PROGRAM PRG_PAOL_02_LightboxScanersCtrl
VAR

	tonEnableCameraSystem				: TON;
	bEnablePackAggregationCameraSystem	: BOOL;
	bEnablePackTriggeringAfterDelayON		: BOOL;

	tofPackAggregationCameraOFFDelay 		: TOF;
	bEnablePackTriggeringAfterDelayOFF		: BOOL;

	fbLightboxLensAirPuls				: FB_Puls;
	tonLightboxLensAirNextBlow		: TON;
	rtrigLightboxLensAirBlowing		: R_TRIG;
	tonLightboxLensAirBlowing		: TOF;
	bPackAggregCameraTrig4Enable			: BOOL;

	fbCameraBoxRead					: FB_3CAM_CameraBoxRead;


	bCameraTriggersArmed			: BOOL;
	bCameraTrigger1Conditioned		: BOOL;
	bCameraTrigger2Conditioned		: BOOL;
	bCameraTrigger3Conditioned		: BOOL;
	bCameraTrigger4Conditioned		: BOOL;

	rtrigCameraTrigger					: ARRAY[0..4] OF R_TRIG;
	aCameraTrigger					: ARRAY[0..4] OF BOOL;
	fbCameraSequenceNo				: FB_3CAM_CameraSequenceNo;

	fbPackScanners_2x5Packs			: FB_3CAM_PackScanners2x5Packs;
	fbPackScanners_3x4Packs			: FB_3CAM_PackScanners3x4Packs;
	fbPackScanners_4x3Packs			: FB_3CAM_PackScanners4x3Packs;
	fbSelectCameraMap				: FB_3CAM_SelectCameraMap;


	fbOUTER_AddNewTriggerID		: FB_PAOL_AddNewTriggerID;
	fbMoveOuterStatusArray			: FB_PACK_MoveOuterStatusArray;	(*Actually is moving OCVPackStatusArray*)

	aPackScanner						: ARRAY[1..3] OF ST_SCANNER_CameraMap;
	fbScannerCtrl						: ARRAY[1..3] OF FB_SCANNER_CameraSelect;
	fbPackCameraEvaluation			: ARRAY[1..3] OF FB_SCANNER_Evaluation;

	fbAddPackCodes					: ARRAY[1..3] OF FB_3CAM_AddPackCodes;

	fbInfeedCamerasSync 				: ARRAY[1..3] OF FB_PAOL_InfeedCamerasSync;

	tonDelayStopOuter					: TON;
	bCameraBufferHighTest 			: BOOL;

	bPackCodeDataInvalid				: BOOL;
	ctuConsecutiveDataInvalid		: CTU;
END_VAR
VAR // added by the converter: edge detectors and wires of the graphical bodies
    _w1, _w3 : BOOL;
    _w2 : UDINT;
END_VAR

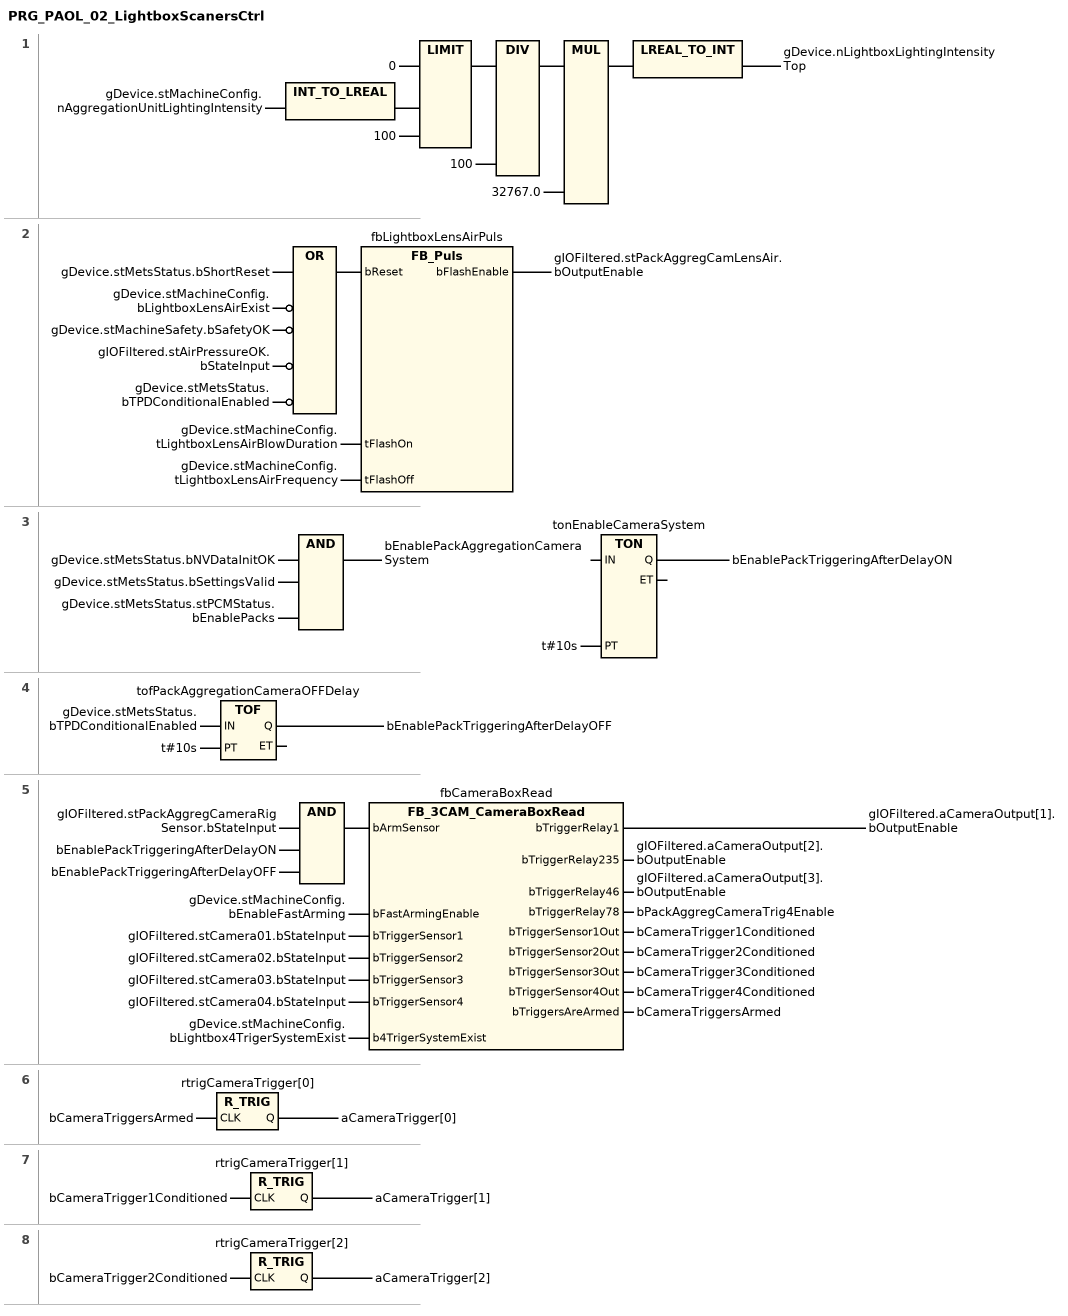
// NETWORK 1
gDevice.nLightboxLightingIntensityTop := LREAL_TO_INT((LIMIT(0, INT_TO_LREAL(gDevice.stMachineConfig.nAggregationUnitLightingIntensity), 100) / 100) * 32767.0);

// NETWORK 2
fbLightboxLensAirPuls(
    bReset := gDevice.stMetsStatus.bShortReset OR NOT gDevice.stMachineConfig.bLightboxLensAirExist OR NOT gDevice.stMachineSafety.bSafetyOK OR NOT gIOFiltered.stAirPressureOK.bStateInput OR NOT gDevice.stMetsStatus.bTPDConditionalEnabled,
    tFlashOn := gDevice.stMachineConfig.tLightboxLensAirBlowDuration,
    tFlashOff := gDevice.stMachineConfig.tLightboxLensAirFrequency); // FB_Puls
gIOFiltered.stPackAggregCamLensAir.bOutputEnable := fbLightboxLensAirPuls.bFlashEnable;

// NETWORK 3
_w1 := gDevice.stMetsStatus.bNVDataInitOK AND gDevice.stMetsStatus.bSettingsValid AND gDevice.stMetsStatus.stPCMStatus.bEnablePacks;
bEnablePackAggregationCameraSystem := _w1;
tonEnableCameraSystem(IN := _w1, PT := t#10s); // TON
bEnablePackTriggeringAfterDelayON := tonEnableCameraSystem.Q;

// NETWORK 4
tofPackAggregationCameraOFFDelay(IN := gDevice.stMetsStatus.bTPDConditionalEnabled, PT := t#10s); // TOF
bEnablePackTriggeringAfterDelayOFF := tofPackAggregationCameraOFFDelay.Q;

// NETWORK 5
fbCameraBoxRead(
    bArmSensor := gIOFiltered.stPackAggregCameraRigSensor.bStateInput AND bEnablePackTriggeringAfterDelayON AND bEnablePackTriggeringAfterDelayOFF,
    bFastArmingEnable := gDevice.stMachineConfig.bEnableFastArming,
    bTriggerSensor1 := gIOFiltered.stCamera01.bStateInput,
    bTriggerSensor2 := gIOFiltered.stCamera02.bStateInput,
    bTriggerSensor3 := gIOFiltered.stCamera03.bStateInput,
    bTriggerSensor4 := gIOFiltered.stCamera04.bStateInput,
    b4TrigerSystemExist := gDevice.stMachineConfig.bLightbox4TrigerSystemExist,
    bTriggerRelay235 => gIOFiltered.aCameraOutput[2].bOutputEnable,
    bTriggerRelay46 => gIOFiltered.aCameraOutput[3].bOutputEnable,
    bTriggerRelay78 => bPackAggregCameraTrig4Enable,
    bTriggerSensor1Out => bCameraTrigger1Conditioned,
    bTriggerSensor2Out => bCameraTrigger2Conditioned,
    bTriggerSensor3Out => bCameraTrigger3Conditioned,
    bTriggerSensor4Out => bCameraTrigger4Conditioned,
    bTriggersAreArmed => bCameraTriggersArmed); // FB_3CAM_CameraBoxRead
gIOFiltered.aCameraOutput[1].bOutputEnable := fbCameraBoxRead.bTriggerRelay1;

// NETWORK 6
rtrigCameraTrigger[0](CLK := bCameraTriggersArmed); // R_TRIG
aCameraTrigger[0] := rtrigCameraTrigger[0].Q;

// NETWORK 7
rtrigCameraTrigger[1](CLK := bCameraTrigger1Conditioned); // R_TRIG
aCameraTrigger[1] := rtrigCameraTrigger[1].Q;

// NETWORK 8
rtrigCameraTrigger[2](CLK := bCameraTrigger2Conditioned); // R_TRIG
aCameraTrigger[2] := rtrigCameraTrigger[2].Q;

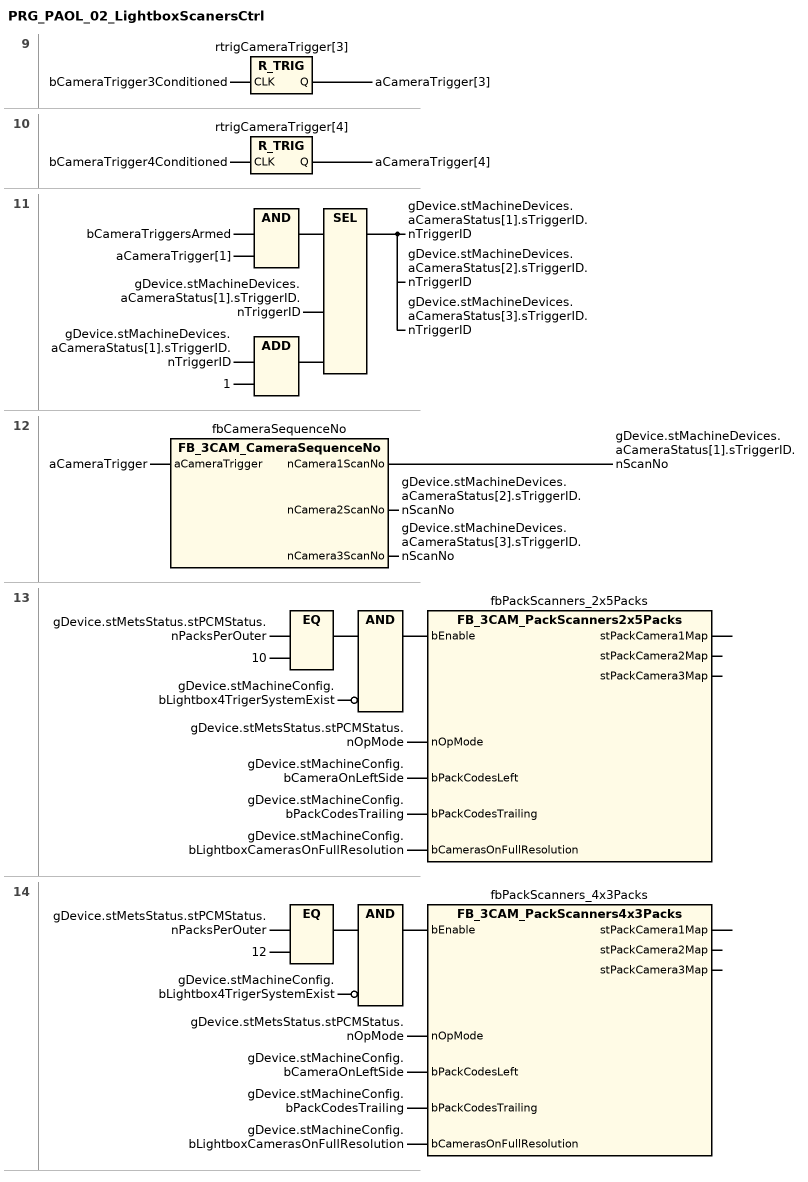
// NETWORK 9
rtrigCameraTrigger[3](CLK := bCameraTrigger3Conditioned); // R_TRIG
aCameraTrigger[3] := rtrigCameraTrigger[3].Q;

// NETWORK 10
rtrigCameraTrigger[4](CLK := bCameraTrigger4Conditioned); // R_TRIG
aCameraTrigger[4] := rtrigCameraTrigger[4].Q;

// NETWORK 11
_w2 := SEL(bCameraTriggersArmed AND aCameraTrigger[1], gDevice.stMachineDevices.aCameraStatus[1].sTriggerID.nTriggerID, gDevice.stMachineDevices.aCameraStatus[1].sTriggerID.nTriggerID + 1);
gDevice.stMachineDevices.aCameraStatus[1].sTriggerID.nTriggerID := _w2;
gDevice.stMachineDevices.aCameraStatus[2].sTriggerID.nTriggerID := _w2;
gDevice.stMachineDevices.aCameraStatus[3].sTriggerID.nTriggerID := _w2;

// NETWORK 12
fbCameraSequenceNo(
    aCameraTrigger := aCameraTrigger,
    nCamera2ScanNo => gDevice.stMachineDevices.aCameraStatus[2].sTriggerID.nScanNo,
    nCamera3ScanNo => gDevice.stMachineDevices.aCameraStatus[3].sTriggerID.nScanNo); // FB_3CAM_CameraSequenceNo
gDevice.stMachineDevices.aCameraStatus[1].sTriggerID.nScanNo := fbCameraSequenceNo.nCamera1ScanNo;

// NETWORK 13
fbPackScanners_2x5Packs(
    bEnable := gDevice.stMetsStatus.stPCMStatus.nPacksPerOuter = 10 AND NOT gDevice.stMachineConfig.bLightbox4TrigerSystemExist,
    nOpMode := gDevice.stMetsStatus.stPCMStatus.nOpMode,
    bPackCodesLeft := gDevice.stMachineConfig.bCameraOnLeftSide,
    bPackCodesTrailing := gDevice.stMachineConfig.bPackCodesTrailing,
    bCamerasOnFullResolution := gDevice.stMachineConfig.bLightboxCamerasOnFullResolution); // FB_3CAM_PackScanners2x5Packs

// NETWORK 14
fbPackScanners_4x3Packs(
    bEnable := gDevice.stMetsStatus.stPCMStatus.nPacksPerOuter = 12 AND NOT gDevice.stMachineConfig.bLightbox4TrigerSystemExist,
    nOpMode := gDevice.stMetsStatus.stPCMStatus.nOpMode,
    bPackCodesLeft := gDevice.stMachineConfig.bCameraOnLeftSide,
    bPackCodesTrailing := gDevice.stMachineConfig.bPackCodesTrailing,
    bCamerasOnFullResolution := gDevice.stMachineConfig.bLightboxCamerasOnFullResolution); // FB_3CAM_PackScanners4x3Packs

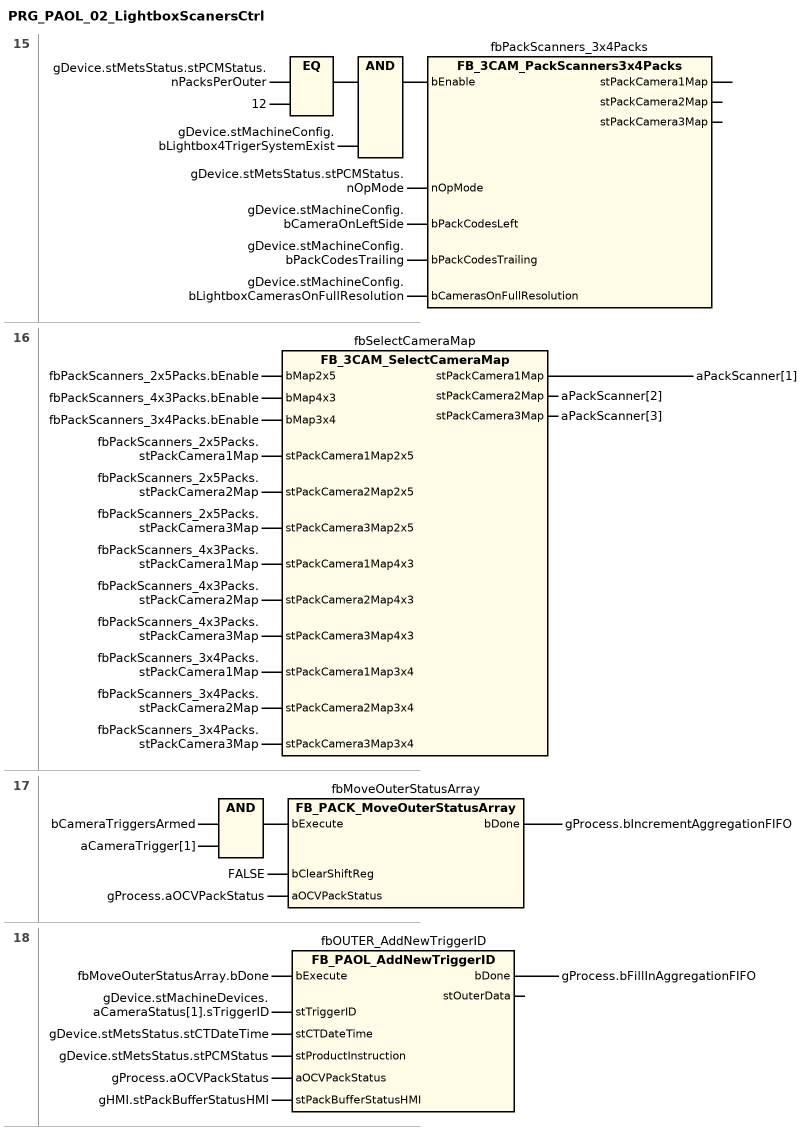
// NETWORK 15
fbPackScanners_3x4Packs(
    bEnable := gDevice.stMetsStatus.stPCMStatus.nPacksPerOuter = 12 AND gDevice.stMachineConfig.bLightbox4TrigerSystemExist,
    nOpMode := gDevice.stMetsStatus.stPCMStatus.nOpMode,
    bPackCodesLeft := gDevice.stMachineConfig.bCameraOnLeftSide,
    bPackCodesTrailing := gDevice.stMachineConfig.bPackCodesTrailing,
    bCamerasOnFullResolution := gDevice.stMachineConfig.bLightboxCamerasOnFullResolution); // FB_3CAM_PackScanners3x4Packs

// NETWORK 16
fbSelectCameraMap(
    bMap2x5 := fbPackScanners_2x5Packs.bEnable,
    bMap4x3 := fbPackScanners_4x3Packs.bEnable,
    bMap3x4 := fbPackScanners_3x4Packs.bEnable,
    stPackCamera1Map2x5 := fbPackScanners_2x5Packs.stPackCamera1Map,
    stPackCamera2Map2x5 := fbPackScanners_2x5Packs.stPackCamera2Map,
    stPackCamera3Map2x5 := fbPackScanners_2x5Packs.stPackCamera3Map,
    stPackCamera1Map4x3 := fbPackScanners_4x3Packs.stPackCamera1Map,
    stPackCamera2Map4x3 := fbPackScanners_4x3Packs.stPackCamera2Map,
    stPackCamera3Map4x3 := fbPackScanners_4x3Packs.stPackCamera3Map,
    stPackCamera1Map3x4 := fbPackScanners_3x4Packs.stPackCamera1Map,
    stPackCamera2Map3x4 := fbPackScanners_3x4Packs.stPackCamera2Map,
    stPackCamera3Map3x4 := fbPackScanners_3x4Packs.stPackCamera3Map,
    stPackCamera2Map => aPackScanner[2],
    stPackCamera3Map => aPackScanner[3]); // FB_3CAM_SelectCameraMap
aPackScanner[1] := fbSelectCameraMap.stPackCamera1Map;

// NETWORK 17
fbMoveOuterStatusArray(
    bExecute := bCameraTriggersArmed AND aCameraTrigger[1],
    bClearShiftReg := FALSE,
    aOCVPackStatus := gProcess.aOCVPackStatus); // FB_PACK_MoveOuterStatusArray
gProcess.bIncrementAggregationFIFO := fbMoveOuterStatusArray.bDone;

// NETWORK 18
fbOUTER_AddNewTriggerID(
    bExecute := fbMoveOuterStatusArray.bDone,
    stTriggerID := gDevice.stMachineDevices.aCameraStatus[1].sTriggerID,
    stCTDateTime := gDevice.stMetsStatus.stCTDateTime,
    stProductInstruction := gDevice.stMetsStatus.stPCMStatus,
    aOCVPackStatus := gProcess.aOCVPackStatus,
    stPackBufferStatusHMI := gHMI.stPackBufferStatusHMI); // FB_PAOL_AddNewTriggerID
gProcess.bFillInAggregationFIFO := fbOUTER_AddNewTriggerID.bDone;

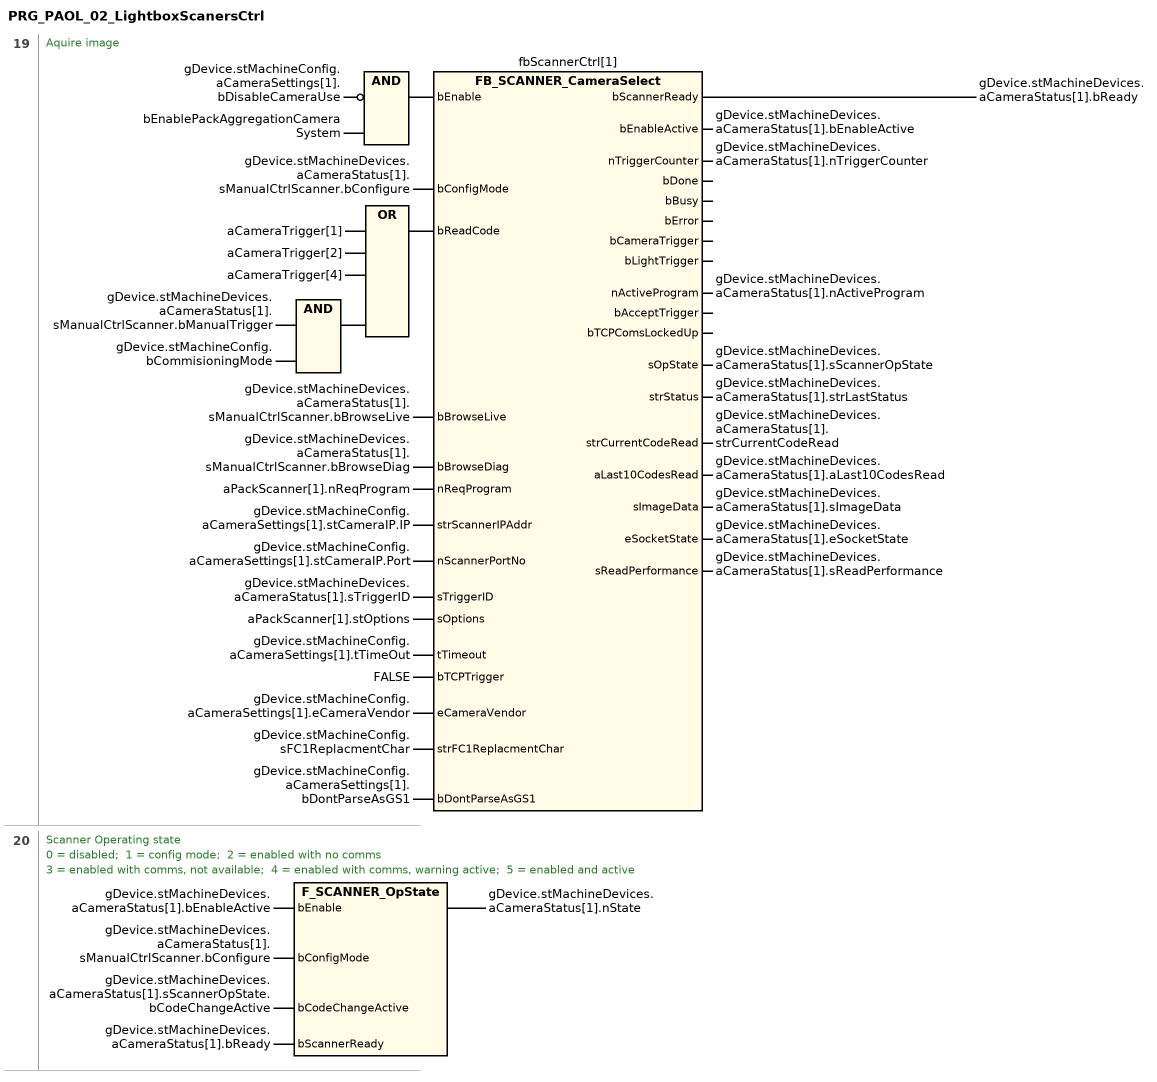
// NETWORK 19
// Aquire image
fbScannerCtrl[1](
    bEnable := NOT gDevice.stMachineConfig.aCameraSettings[1].bDisableCameraUse AND bEnablePackAggregationCameraSystem,
    bConfigMode := gDevice.stMachineDevices.aCameraStatus[1].sManualCtrlScanner.bConfigure,
    bReadCode := aCameraTrigger[1] OR aCameraTrigger[2] OR aCameraTrigger[4] OR gDevice.stMachineDevices.aCameraStatus[1].sManualCtrlScanner.bManualTrigger AND gDevice.stMachineConfig.bCommisioningMode,
    bBrowseLive := gDevice.stMachineDevices.aCameraStatus[1].sManualCtrlScanner.bBrowseLive,
    bBrowseDiag := gDevice.stMachineDevices.aCameraStatus[1].sManualCtrlScanner.bBrowseDiag,
    nReqProgram := aPackScanner[1].nReqProgram,
    strScannerIPAddr := gDevice.stMachineConfig.aCameraSettings[1].stCameraIP.IP,
    nScannerPortNo := gDevice.stMachineConfig.aCameraSettings[1].stCameraIP.Port,
    sTriggerID := gDevice.stMachineDevices.aCameraStatus[1].sTriggerID,
    sOptions := aPackScanner[1].stOptions,
    tTimeout := gDevice.stMachineConfig.aCameraSettings[1].tTimeOut,
    bTCPTrigger := FALSE,
    eCameraVendor := gDevice.stMachineConfig.aCameraSettings[1].eCameraVendor,
    strFC1ReplacmentChar := gDevice.stMachineConfig.sFC1ReplacmentChar,
    bDontParseAsGS1 := gDevice.stMachineConfig.aCameraSettings[1].bDontParseAsGS1,
    bEnableActive => gDevice.stMachineDevices.aCameraStatus[1].bEnableActive,
    nTriggerCounter => gDevice.stMachineDevices.aCameraStatus[1].nTriggerCounter,
    nActiveProgram => gDevice.stMachineDevices.aCameraStatus[1].nActiveProgram,
    sOpState => gDevice.stMachineDevices.aCameraStatus[1].sScannerOpState,
    strStatus => gDevice.stMachineDevices.aCameraStatus[1].strLastStatus,
    strCurrentCodeRead => gDevice.stMachineDevices.aCameraStatus[1].strCurrentCodeRead,
    aLast10CodesRead => gDevice.stMachineDevices.aCameraStatus[1].aLast10CodesRead,
    sImageData => gDevice.stMachineDevices.aCameraStatus[1].sImageData,
    eSocketState => gDevice.stMachineDevices.aCameraStatus[1].eSocketState,
    sReadPerformance => gDevice.stMachineDevices.aCameraStatus[1].sReadPerformance); // FB_SCANNER_CameraSelect
gDevice.stMachineDevices.aCameraStatus[1].bReady := fbScannerCtrl[1].bScannerReady;

// NETWORK 20
// 					Scanner Operating state
// 0 = disabled;  1 = config mode;  2 = enabled with no comms
// 3 = enabled with comms, not available;  4 = enabled with comms, warning active;  5 = enabled and active
//
gDevice.stMachineDevices.aCameraStatus[1].nState := F_SCANNER_OpState(bEnable := gDevice.stMachineDevices.aCameraStatus[1].bEnableActive, bConfigMode := gDevice.stMachineDevices.aCameraStatus[1].sManualCtrlScanner.bConfigure, bCodeChangeActive := gDevice.stMachineDevices.aCameraStatus[1].sScannerOpState.bCodeChangeActive, bScannerReady := gDevice.stMachineDevices.aCameraStatus[1].bReady);

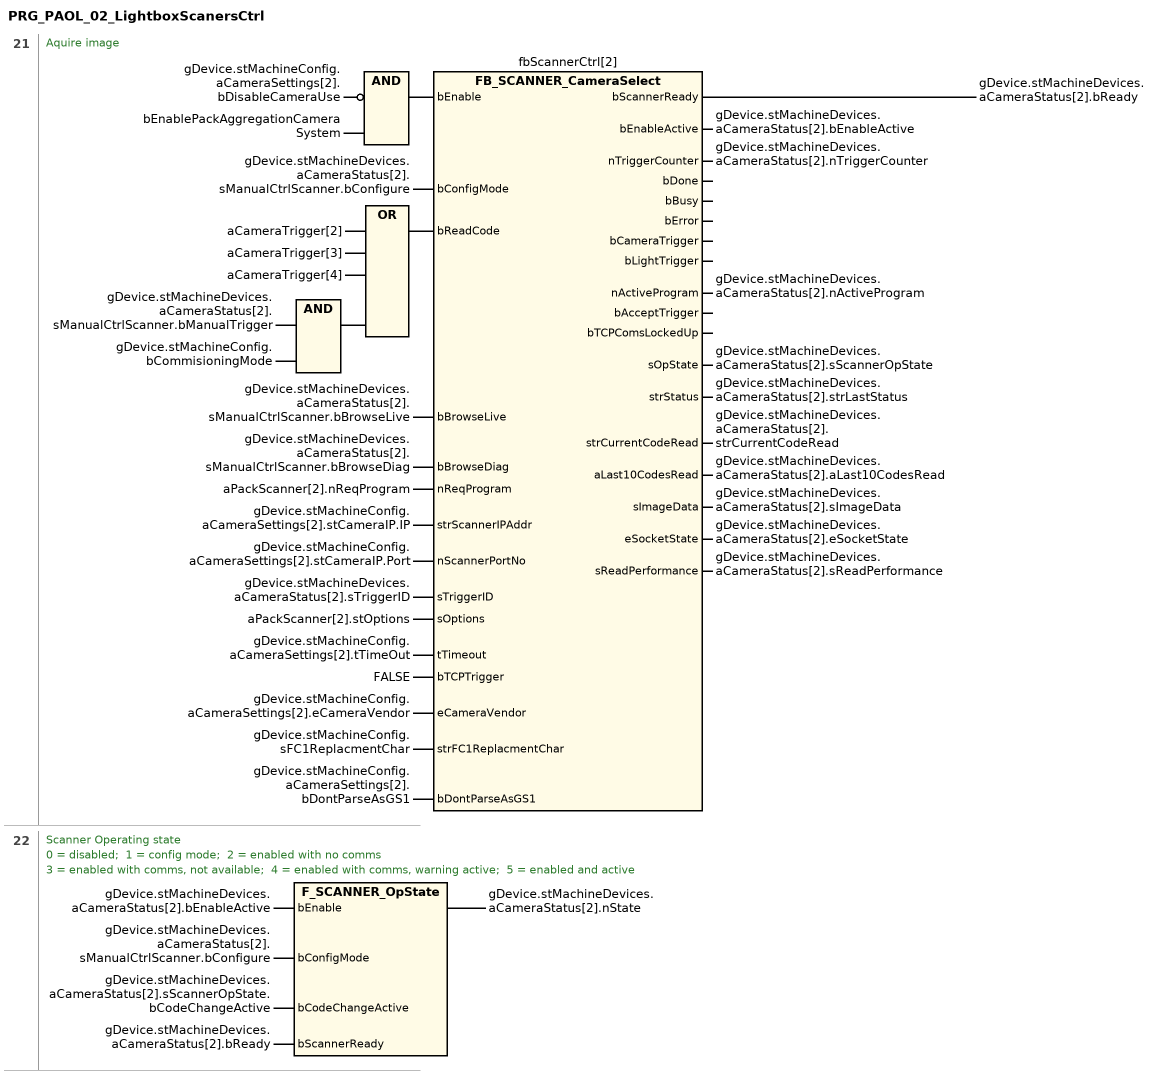
// NETWORK 21
// Aquire image
fbScannerCtrl[2](
    bEnable := NOT gDevice.stMachineConfig.aCameraSettings[2].bDisableCameraUse AND bEnablePackAggregationCameraSystem,
    bConfigMode := gDevice.stMachineDevices.aCameraStatus[2].sManualCtrlScanner.bConfigure,
    bReadCode := aCameraTrigger[2] OR aCameraTrigger[3] OR aCameraTrigger[4] OR gDevice.stMachineDevices.aCameraStatus[2].sManualCtrlScanner.bManualTrigger AND gDevice.stMachineConfig.bCommisioningMode,
    bBrowseLive := gDevice.stMachineDevices.aCameraStatus[2].sManualCtrlScanner.bBrowseLive,
    bBrowseDiag := gDevice.stMachineDevices.aCameraStatus[2].sManualCtrlScanner.bBrowseDiag,
    nReqProgram := aPackScanner[2].nReqProgram,
    strScannerIPAddr := gDevice.stMachineConfig.aCameraSettings[2].stCameraIP.IP,
    nScannerPortNo := gDevice.stMachineConfig.aCameraSettings[2].stCameraIP.Port,
    sTriggerID := gDevice.stMachineDevices.aCameraStatus[2].sTriggerID,
    sOptions := aPackScanner[2].stOptions,
    tTimeout := gDevice.stMachineConfig.aCameraSettings[2].tTimeOut,
    bTCPTrigger := FALSE,
    eCameraVendor := gDevice.stMachineConfig.aCameraSettings[2].eCameraVendor,
    strFC1ReplacmentChar := gDevice.stMachineConfig.sFC1ReplacmentChar,
    bDontParseAsGS1 := gDevice.stMachineConfig.aCameraSettings[2].bDontParseAsGS1,
    bEnableActive => gDevice.stMachineDevices.aCameraStatus[2].bEnableActive,
    nTriggerCounter => gDevice.stMachineDevices.aCameraStatus[2].nTriggerCounter,
    nActiveProgram => gDevice.stMachineDevices.aCameraStatus[2].nActiveProgram,
    sOpState => gDevice.stMachineDevices.aCameraStatus[2].sScannerOpState,
    strStatus => gDevice.stMachineDevices.aCameraStatus[2].strLastStatus,
    strCurrentCodeRead => gDevice.stMachineDevices.aCameraStatus[2].strCurrentCodeRead,
    aLast10CodesRead => gDevice.stMachineDevices.aCameraStatus[2].aLast10CodesRead,
    sImageData => gDevice.stMachineDevices.aCameraStatus[2].sImageData,
    eSocketState => gDevice.stMachineDevices.aCameraStatus[2].eSocketState,
    sReadPerformance => gDevice.stMachineDevices.aCameraStatus[2].sReadPerformance); // FB_SCANNER_CameraSelect
gDevice.stMachineDevices.aCameraStatus[2].bReady := fbScannerCtrl[2].bScannerReady;

// NETWORK 22
// 					Scanner Operating state
// 0 = disabled;  1 = config mode;  2 = enabled with no comms
// 3 = enabled with comms, not available;  4 = enabled with comms, warning active;  5 = enabled and active
//
gDevice.stMachineDevices.aCameraStatus[2].nState := F_SCANNER_OpState(bEnable := gDevice.stMachineDevices.aCameraStatus[2].bEnableActive, bConfigMode := gDevice.stMachineDevices.aCameraStatus[2].sManualCtrlScanner.bConfigure, bCodeChangeActive := gDevice.stMachineDevices.aCameraStatus[2].sScannerOpState.bCodeChangeActive, bScannerReady := gDevice.stMachineDevices.aCameraStatus[2].bReady);

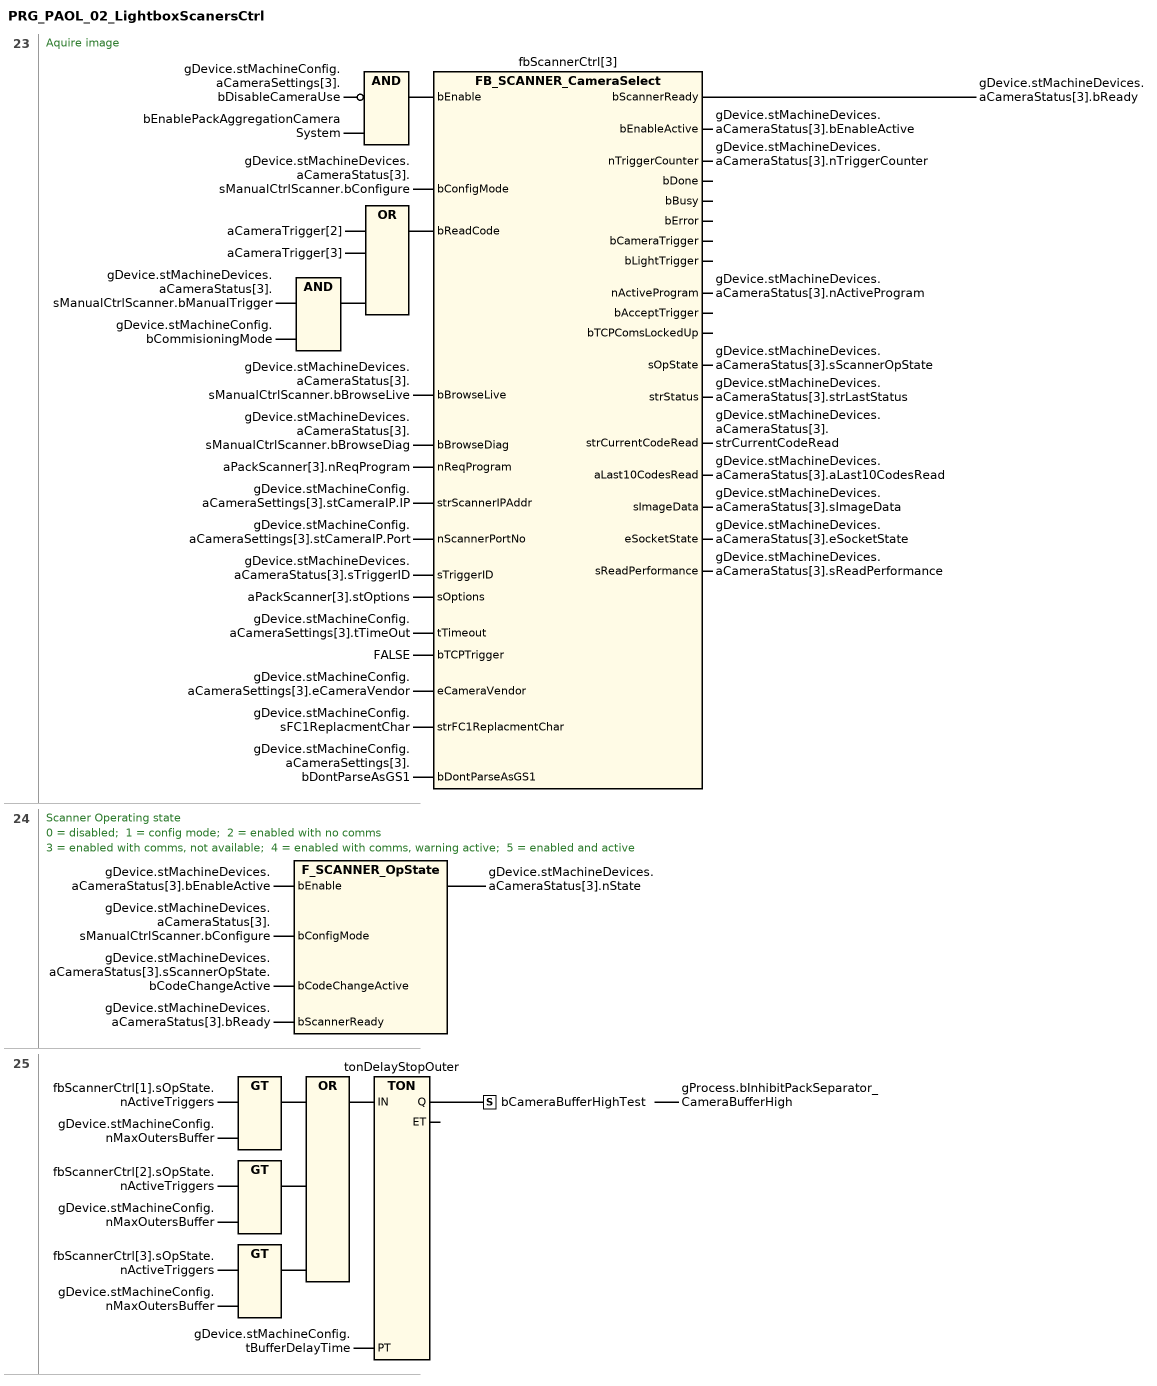
// NETWORK 23
// Aquire image
fbScannerCtrl[3](
    bEnable := NOT gDevice.stMachineConfig.aCameraSettings[3].bDisableCameraUse AND bEnablePackAggregationCameraSystem,
    bConfigMode := gDevice.stMachineDevices.aCameraStatus[3].sManualCtrlScanner.bConfigure,
    bReadCode := aCameraTrigger[2] OR aCameraTrigger[3] OR gDevice.stMachineDevices.aCameraStatus[3].sManualCtrlScanner.bManualTrigger AND gDevice.stMachineConfig.bCommisioningMode,
    bBrowseLive := gDevice.stMachineDevices.aCameraStatus[3].sManualCtrlScanner.bBrowseLive,
    bBrowseDiag := gDevice.stMachineDevices.aCameraStatus[3].sManualCtrlScanner.bBrowseDiag,
    nReqProgram := aPackScanner[3].nReqProgram,
    strScannerIPAddr := gDevice.stMachineConfig.aCameraSettings[3].stCameraIP.IP,
    nScannerPortNo := gDevice.stMachineConfig.aCameraSettings[3].stCameraIP.Port,
    sTriggerID := gDevice.stMachineDevices.aCameraStatus[3].sTriggerID,
    sOptions := aPackScanner[3].stOptions,
    tTimeout := gDevice.stMachineConfig.aCameraSettings[3].tTimeOut,
    bTCPTrigger := FALSE,
    eCameraVendor := gDevice.stMachineConfig.aCameraSettings[3].eCameraVendor,
    strFC1ReplacmentChar := gDevice.stMachineConfig.sFC1ReplacmentChar,
    bDontParseAsGS1 := gDevice.stMachineConfig.aCameraSettings[3].bDontParseAsGS1,
    bEnableActive => gDevice.stMachineDevices.aCameraStatus[3].bEnableActive,
    nTriggerCounter => gDevice.stMachineDevices.aCameraStatus[3].nTriggerCounter,
    nActiveProgram => gDevice.stMachineDevices.aCameraStatus[3].nActiveProgram,
    sOpState => gDevice.stMachineDevices.aCameraStatus[3].sScannerOpState,
    strStatus => gDevice.stMachineDevices.aCameraStatus[3].strLastStatus,
    strCurrentCodeRead => gDevice.stMachineDevices.aCameraStatus[3].strCurrentCodeRead,
    aLast10CodesRead => gDevice.stMachineDevices.aCameraStatus[3].aLast10CodesRead,
    sImageData => gDevice.stMachineDevices.aCameraStatus[3].sImageData,
    eSocketState => gDevice.stMachineDevices.aCameraStatus[3].eSocketState,
    sReadPerformance => gDevice.stMachineDevices.aCameraStatus[3].sReadPerformance); // FB_SCANNER_CameraSelect
gDevice.stMachineDevices.aCameraStatus[3].bReady := fbScannerCtrl[3].bScannerReady;

// NETWORK 24
// 					Scanner Operating state
// 0 = disabled;  1 = config mode;  2 = enabled with no comms
// 3 = enabled with comms, not available;  4 = enabled with comms, warning active;  5 = enabled and active
//
gDevice.stMachineDevices.aCameraStatus[3].nState := F_SCANNER_OpState(bEnable := gDevice.stMachineDevices.aCameraStatus[3].bEnableActive, bConfigMode := gDevice.stMachineDevices.aCameraStatus[3].sManualCtrlScanner.bConfigure, bCodeChangeActive := gDevice.stMachineDevices.aCameraStatus[3].sScannerOpState.bCodeChangeActive, bScannerReady := gDevice.stMachineDevices.aCameraStatus[3].bReady);

// NETWORK 25
tonDelayStopOuter(IN := fbScannerCtrl[1].sOpState.nActiveTriggers > gDevice.stMachineConfig.nMaxOutersBuffer OR fbScannerCtrl[2].sOpState.nActiveTriggers > gDevice.stMachineConfig.nMaxOutersBuffer OR fbScannerCtrl[3].sOpState.nActiveTriggers > gDevice.stMachineConfig.nMaxOutersBuffer, PT := gDevice.stMachineConfig.tBufferDelayTime); // TON
bCameraBufferHighTest S= tonDelayStopOuter.Q;
gProcess.bInhibitPackSeparator_CameraBufferHigh := tonDelayStopOuter.Q;

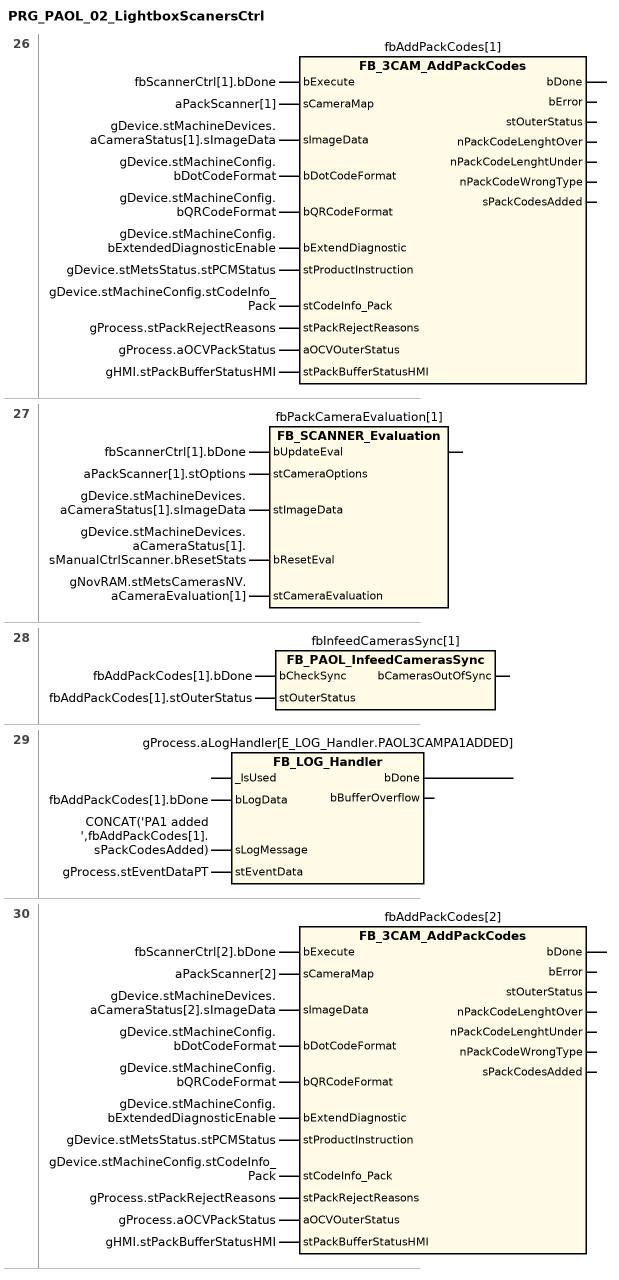
// NETWORK 26
fbAddPackCodes[1](
    bExecute := fbScannerCtrl[1].bDone,
    sCameraMap := aPackScanner[1],
    sImageData := gDevice.stMachineDevices.aCameraStatus[1].sImageData,
    bDotCodeFormat := gDevice.stMachineConfig.bDotCodeFormat,
    bQRCodeFormat := gDevice.stMachineConfig.bQRCodeFormat,
    bExtendDiagnostic := gDevice.stMachineConfig.bExtendedDiagnosticEnable,
    stProductInstruction := gDevice.stMetsStatus.stPCMStatus,
    stCodeInfo_Pack := gDevice.stMachineConfig.stCodeInfo_Pack,
    stPackRejectReasons := gProcess.stPackRejectReasons,
    aOCVOuterStatus := gProcess.aOCVPackStatus,
    stPackBufferStatusHMI := gHMI.stPackBufferStatusHMI); // FB_3CAM_AddPackCodes

// NETWORK 27
fbPackCameraEvaluation[1](
    bUpdateEval := fbScannerCtrl[1].bDone,
    stCameraOptions := aPackScanner[1].stOptions,
    stImageData := gDevice.stMachineDevices.aCameraStatus[1].sImageData,
    bResetEval := gDevice.stMachineDevices.aCameraStatus[1].sManualCtrlScanner.bResetStats,
    stCameraEvaluation := gNovRAM.stMetsCamerasNV.aCameraEvaluation[1]); // FB_SCANNER_Evaluation

// NETWORK 28
fbInfeedCamerasSync[1](bCheckSync := fbAddPackCodes[1].bDone, stOuterStatus := fbAddPackCodes[1].stOuterStatus); // FB_PAOL_InfeedCamerasSync

// NETWORK 29
gProcess.aLogHandler[E_LOG_Handler.PAOL3CAMPA1ADDED](
    bLogData := fbAddPackCodes[1].bDone,
    sLogMessage := CONCAT('PA1 added ',fbAddPackCodes[1].sPackCodesAdded),
    stEventData := gProcess.stEventDataPT); // FB_LOG_Handler

// NETWORK 30
fbAddPackCodes[2](
    bExecute := fbScannerCtrl[2].bDone,
    sCameraMap := aPackScanner[2],
    sImageData := gDevice.stMachineDevices.aCameraStatus[2].sImageData,
    bDotCodeFormat := gDevice.stMachineConfig.bDotCodeFormat,
    bQRCodeFormat := gDevice.stMachineConfig.bQRCodeFormat,
    bExtendDiagnostic := gDevice.stMachineConfig.bExtendedDiagnosticEnable,
    stProductInstruction := gDevice.stMetsStatus.stPCMStatus,
    stCodeInfo_Pack := gDevice.stMachineConfig.stCodeInfo_Pack,
    stPackRejectReasons := gProcess.stPackRejectReasons,
    aOCVOuterStatus := gProcess.aOCVPackStatus,
    stPackBufferStatusHMI := gHMI.stPackBufferStatusHMI); // FB_3CAM_AddPackCodes

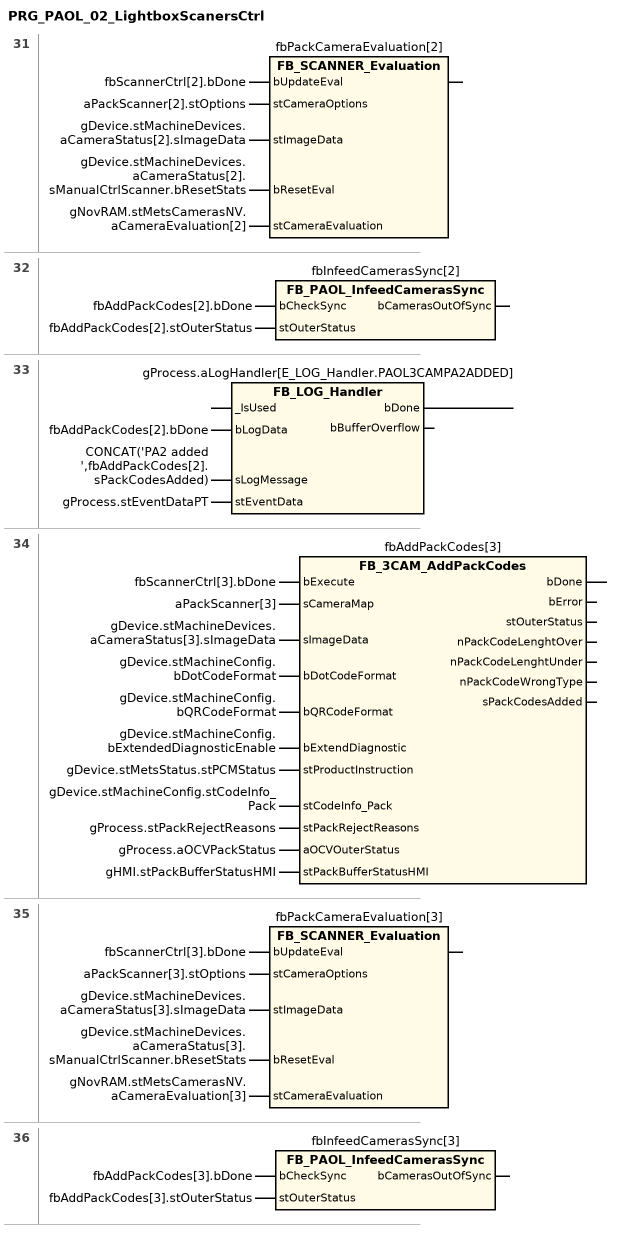
// NETWORK 31
fbPackCameraEvaluation[2](
    bUpdateEval := fbScannerCtrl[2].bDone,
    stCameraOptions := aPackScanner[2].stOptions,
    stImageData := gDevice.stMachineDevices.aCameraStatus[2].sImageData,
    bResetEval := gDevice.stMachineDevices.aCameraStatus[2].sManualCtrlScanner.bResetStats,
    stCameraEvaluation := gNovRAM.stMetsCamerasNV.aCameraEvaluation[2]); // FB_SCANNER_Evaluation

// NETWORK 32
fbInfeedCamerasSync[2](bCheckSync := fbAddPackCodes[2].bDone, stOuterStatus := fbAddPackCodes[2].stOuterStatus); // FB_PAOL_InfeedCamerasSync

// NETWORK 33
gProcess.aLogHandler[E_LOG_Handler.PAOL3CAMPA2ADDED](
    bLogData := fbAddPackCodes[2].bDone,
    sLogMessage := CONCAT('PA2 added ',fbAddPackCodes[2].sPackCodesAdded),
    stEventData := gProcess.stEventDataPT); // FB_LOG_Handler

// NETWORK 34
fbAddPackCodes[3](
    bExecute := fbScannerCtrl[3].bDone,
    sCameraMap := aPackScanner[3],
    sImageData := gDevice.stMachineDevices.aCameraStatus[3].sImageData,
    bDotCodeFormat := gDevice.stMachineConfig.bDotCodeFormat,
    bQRCodeFormat := gDevice.stMachineConfig.bQRCodeFormat,
    bExtendDiagnostic := gDevice.stMachineConfig.bExtendedDiagnosticEnable,
    stProductInstruction := gDevice.stMetsStatus.stPCMStatus,
    stCodeInfo_Pack := gDevice.stMachineConfig.stCodeInfo_Pack,
    stPackRejectReasons := gProcess.stPackRejectReasons,
    aOCVOuterStatus := gProcess.aOCVPackStatus,
    stPackBufferStatusHMI := gHMI.stPackBufferStatusHMI); // FB_3CAM_AddPackCodes

// NETWORK 35
fbPackCameraEvaluation[3](
    bUpdateEval := fbScannerCtrl[3].bDone,
    stCameraOptions := aPackScanner[3].stOptions,
    stImageData := gDevice.stMachineDevices.aCameraStatus[3].sImageData,
    bResetEval := gDevice.stMachineDevices.aCameraStatus[3].sManualCtrlScanner.bResetStats,
    stCameraEvaluation := gNovRAM.stMetsCamerasNV.aCameraEvaluation[3]); // FB_SCANNER_Evaluation

// NETWORK 36
fbInfeedCamerasSync[3](bCheckSync := fbAddPackCodes[3].bDone, stOuterStatus := fbAddPackCodes[3].stOuterStatus); // FB_PAOL_InfeedCamerasSync

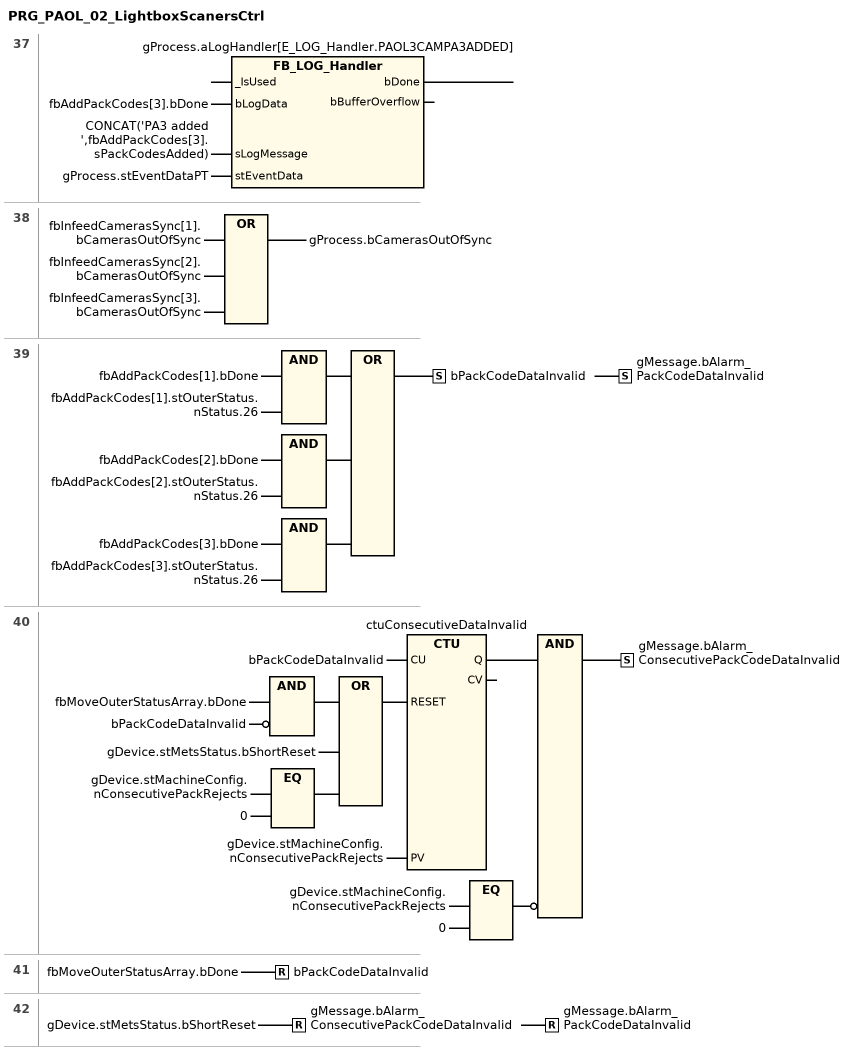
// NETWORK 37
gProcess.aLogHandler[E_LOG_Handler.PAOL3CAMPA3ADDED](
    bLogData := fbAddPackCodes[3].bDone,
    sLogMessage := CONCAT('PA3 added ',fbAddPackCodes[3].sPackCodesAdded),
    stEventData := gProcess.stEventDataPT); // FB_LOG_Handler

// NETWORK 38
gProcess.bCamerasOutOfSync := fbInfeedCamerasSync[1].bCamerasOutOfSync OR fbInfeedCamerasSync[2].bCamerasOutOfSync OR fbInfeedCamerasSync[3].bCamerasOutOfSync;

// NETWORK 39
_w3 := fbAddPackCodes[1].bDone AND fbAddPackCodes[1].stOuterStatus.nStatus.26 OR fbAddPackCodes[2].bDone AND fbAddPackCodes[2].stOuterStatus.nStatus.26 OR fbAddPackCodes[3].bDone AND fbAddPackCodes[3].stOuterStatus.nStatus.26;
bPackCodeDataInvalid S= _w3;
gMessage.bAlarm_PackCodeDataInvalid S= _w3;

// NETWORK 40
ctuConsecutiveDataInvalid(
    CU := bPackCodeDataInvalid,
    RESET := fbMoveOuterStatusArray.bDone AND NOT bPackCodeDataInvalid OR gDevice.stMetsStatus.bShortReset OR gDevice.stMachineConfig.nConsecutivePackRejects = 0,
    PV := gDevice.stMachineConfig.nConsecutivePackRejects); // CTU
gMessage.bAlarm_ConsecutivePackCodeDataInvalid S= ctuConsecutiveDataInvalid.Q AND NOT (gDevice.stMachineConfig.nConsecutivePackRejects = 0);

// NETWORK 41
bPackCodeDataInvalid R= fbMoveOuterStatusArray.bDone;

// NETWORK 42
gMessage.bAlarm_ConsecutivePackCodeDataInvalid R= gDevice.stMetsStatus.bShortReset;
gMessage.bAlarm_PackCodeDataInvalid R= gDevice.stMetsStatus.bShortReset;

END_PROGRAM

(* stored: Version 1.1.0.1
   POU PRG_PAOL_02_LightboxScanersCtrl: Id {b7a16d25-788d-4097-ba6b-0542917af820}, SpecialFunc None *)
